FUNCTION_BLOCK FB_VFD_ABB_ACS480 EXTENDS FB_UniversalVFDModbus

VAR
	VFD_CTRL_RUN_EMERGENCY_STOP : WORD;
	TempData0: U_Word2Int;
END_VAR

SUPER^();

METHOD Convert : BOOL
VAR_INPUT
	iRegionNo	:	INT;
	pReadData	:	POINTER TO word;
END_VAR
CASE	iRegionNo OF

	0: // status
		IF pReadData[0].15 = TRUE THEN
			eVfdStatus := VFD_STATUS_FAULT;
			
		ELSIF (eVfdState = VFD_INITIALIZING
			OR eVfdState = VFD_READY_INITIALIZED)
			AND pReadData[0].0 = TRUE
			AND pReadData[0].1 = TRUE	
			AND pReadData[0].2 = TRUE
			THEN
			eVfdStatus :=  VFD_STATUS_READY_TO_RUN;
				
		ELSIF pReadData[0].3 = FALSE THEN
			eVfdStatus :=  VFD_STATUS_STOP;
			
		ELSIF pReadData[0].3 = TRUE	//run
			AND pReadData[0].10 = FALSE	// Drive reference is in the forward direction	
			AND pReadData[0].11 = FALSE//Drive is running in the forward direction
			THEN		
			eVfdStatus := VFD_STATUS_RUNNING_FORWARD;
		
		ELSIF pReadData[0].3 = TRUE	//run
			AND pReadData[0].10 = TRUE	// Drive reference is in the forward direction	
			AND pReadData[0].11 = TRUE//Drive is running in the forward direction
			THEN		
			eVfdStatus := VFD_STATUS_RUNNING_REVERSE;
		
		END_IF
	1: 
		TempData0.iWord := pReadData[0];
		lrHzActual		:= ABS(INT_TO_LREAL( TempData0.iInt)*0.0025);//50/20000;	
		lrCurrent		:= WORD_TO_LREAL( pReadData[1])*0.01;	//46.05 = 100
		lrDcVoltage		:= WORD_TO_LREAL( pReadData[5])*0.1;	
	
	2: 
		lrVacOutToMotor	:= WORD_TO_LREAL( pReadData[0]);	//4099	/1
		lrPowerKw		:= WORD_TO_LREAL( pReadData[1])*0.01;		//46.04
	
	3:
		lrTotalKwh :=  WORD_TO_LREAL( pReadData[0])*0.1;
		
	4: 
		lrSpeed :=  WORD_TO_LREAL( pReadData[0]);
	
	


END_CASE
END_METHOD

METHOD  FirstCycle 
VAR_INPUT
	sName : STRING;
	iUnitID : BYTE ; // modbus address of the device : 1- 255
END_VAR
SUPER^.FirstCycle( sName := sName, iUnitID := iUnitID);
(*Assign Ctrol Word : user Manual M-driver*)
VFD_CTRL_RESET_FAULT := 2#0001_0001;
VFD_CTRL_RUN_FORWARD := 2#0000_0010;
VFD_CTRL_RUN_REVERSE := 2#0000_0110;
VFD_CTRL_STOP_FREE 	 := 2#0010_0000_0001;
VFD_CTRL_STOP_SPEED_DOWN := 2#1000_0001;
VFD_CTRL_RUN_EMERGENCY_STOP := 2#0001_0000_0001;

// actual state	
	arrAddressRead[0][0] := 3;
	arrAddressRead[0][1] := 1;
	arrAddressRead[0][2] := E_ModbusFunction.ReadHoldingRegisters;

//mode0 address = 40000 + function*100 + sub function -1
	// actual hz  
	arrAddressRead[1][0] := 105; // 01.06
	arrAddressRead[1][1] := 6;
	arrAddressRead[1][2] := E_ModbusFunction.ReadHoldingRegisters;
	
	arrAddressRead[2][0] := 112; // 01.13
	arrAddressRead[2][1] := 2;
	arrAddressRead[2][2] := E_ModbusFunction.ReadHoldingRegisters;
	
	arrAddressRead[3][0] := 119; // 01.20
	arrAddressRead[3][1] := 1;
	arrAddressRead[3][2] := E_ModbusFunction.ReadHoldingRegisters;
	
	arrAddressRead[4][0] := 101; // 01.20
	arrAddressRead[4][1] := 1;
	arrAddressRead[4][2] := E_ModbusFunction.ReadHoldingRegisters;
iNumAddRegionRead	:= 5;

/////write control WORD VFD, // use ctrol word and frequency in 1 modbus write
arrAddressWrite[iCTRL_WORD][0]	:= 0;
arrAddressWrite[iCTRL_WORD][1]	:= 2;
arrAddressWrite[iCTRL_WORD][2]	:= VFD_CTRL_STOP_FREE;
arrAddressWrite[iCTRL_WORD][10]	:= E_ModbusFunction.WriteMultipleRegisters;

// Frequency
//arrAddressWrite[iCTRL_FREQUENCY_WORD][0]	:= 1;
//arrAddressWrite[iCTRL_FREQUENCY_WORD][1]	:= 1;
							(*MUST BE CARE FULL WHEN USE FLOATING POINT CONVERT*)
arrAddressWrite[iCTRL_FREQUENCY_WORD][3]	:= LREAL_TO_WORD( F_ScaleValue(	rangeRawMin := 0,
																				rangeRawMax := 50,
																				RangeScaleMin :=0,
																				RangeScaleMax := 20000,
																				ValueRaw := 0)
										  );
										  
iNumAddRegionWrite := 1;// use ctrol word and frequency in 1 modbus write
END_METHOD

METHOD PROTECTED  MS_Aborting
arrAddressWrite[iCTRL_WORD][2]	:= VFD_CTRL_STOP_FREE;
SUPER^.MS_Aborting();
END_METHOD

METHOD  PROTECTED  MS_Initializing
SUPER^.MS_Initializing();
END_METHOD

METHOD PROTECTED  MS_RunForward
VAR_INPUT
END_VAR
// use ctrol word and frequency in 1 modbus write WRITE MULTIES REGIS
arrAddressWrite[iCTRL_WORD][3] :=  LREAL_TO_WORD( 
															F_ScaleValue(	rangeRawMin := 0,
																			rangeRawMax := 50,
																			RangeScaleMin := 0,
																			RangeScaleMax := 20000,
																			ValueRaw := lrHzControl) 
																				);
SUPER^.MS_RunForward();
END_METHOD

METHOD PROTECTED  MS_RunReverse
VAR_INPUT
END_VAR
// use ctrol word and frequency in 1 modbus write WRITE MULTIES REGIS
arrAddressWrite[iCTRL_WORD][3] :=  LREAL_TO_WORD( 
															F_ScaleValue(	rangeRawMin := 0,
																			rangeRawMax := 50,
																			RangeScaleMin := 0,
																			RangeScaleMax := 20000,
																			ValueRaw := lrHzControl) 
																				);
SUPER^.MS_RunReverse();
END_METHOD

END_FUNCTION_BLOCK

(* stored: Version 1.1.0.1, ProductVersion 3.1.4024.12
   POU FB_VFD_ABB_ACS480: Id {96595415-751d-464c-bab2-749904d5515d}, SpecialFunc None
   Method Convert: Id {38687b8c-f3a1-4fab-8feb-ea3ee5eed31d}
   Method FirstCycle: Id {3ae3af73-66a5-4fe8-bb9c-cf2fccd9f358}
   Method MS_Aborting: Id {4b3b5df2-b4fb-4af1-b70d-bb31381aceb2}
   Method MS_Initializing: Id {e68f7a5b-7f0f-475c-b606-f65058277e1e}
   Method MS_RunForward: Id {dfb441b6-3fe3-4262-9d67-6a331974a3c0}
   Method MS_RunReverse: Id {9c92e45f-7e6a-4daa-961b-df03857394f0} *)
